TYPE ST115_PnpHorPos_e : ST110_PnpHorPos_e;
END_TYPE

(* stored: Version 1.1.0.1, ProductVersion 3.1.4024.6
   DUT ST115_PnpHorPos_e: Id {e614e949-788f-4541-8448-ff229b39baa4} *)
